// TIA Portal V20 export
DATA_BLOCK "DB_LoaderAxis"   // DB206
// stored: AutoNumber false, InstanceOfName FB_LoaderAxis, InstanceOfType FB
"FB_LoaderAxis"
   // VAR_INPUT
   //    iPLCModeReq : Bool;
   //    iCNCModeReq : Bool;
   //    iU1StartReq : Bool;
   //    iU2StartReq : Bool;
   //    iVStartReq : Bool;
   //    iWStartReq : Bool;
   //    iU1PosSetPoint : Real;
   //    iU2PosSetPoint : Real;
   //    iVPosSetPoint : Real;
   //    iWPosSetPoint : Real;
   // END_VAR
   // VAR_OUTPUT
   //    oU1InPos : Bool;
   //    oU2InPos : Bool;
   //    oVInPos : Bool;
   //    oWInPos : Bool;
   // END_VAR
   // VAR
   //    sAxisPLCMode : Bool;
   //    sAxisCNCMode : Bool;
   //    sAllAxisPLCMode : Bool;
   //    sAllAxisCNCMode : Bool;
   //    sU1StartMove : Bool;
   //    sU2StartMove : Bool;
   //    sVStartMove : Bool;
   //    sWStartMove : Bool;
   //    sU1MoveError : Bool;
   //    sU2MoveError : Bool;
   //    sVMoveError : Bool;
   //    sWMoveError : Bool;
   //    sU1InPos : Bool;
   //    sU2InPos : Bool;
   //    sVInPos : Bool;
   //    sWInPos : Bool;
   //    sU1SetPos : Real;
   //    sU2SetPos : Real;
   //    sVSetPos : Real;
   //    sWSetPos : Real;
   //    sU1MoveState : Byte;
   //    sU2MoveState : Byte;
   //    sVMoveState : Byte;
   //    sWMoveState : Byte;
   //    sU1ActFeedRate : LReal;
   //    sU2ActFeedRate : LReal;
   //    sVActFeedRate : LReal;
   //    sWActFeedRate : LReal;
   //    sU1DrivedByPLC : Bool;
   //    sU2DrivedByPLC : Bool;
   //    sVDrivedByPLC : Bool;
   //    sWDrivedByPLC : Bool;
   //    sU1Positioning { ExternalAccessible := 'False'; ExternalVisible := 'False'; ExternalWritable := 'False'} : Bool;
   //    sU2Positioning { ExternalAccessible := 'False'; ExternalVisible := 'False'; ExternalWritable := 'False'} : Bool;
   //    sVPositioning { ExternalAccessible := 'False'; ExternalVisible := 'False'; ExternalWritable := 'False'} : Bool;
   //    sWPositioning { ExternalAccessible := 'False'; ExternalVisible := 'False'; ExternalWritable := 'False'} : Bool;
   //    sFeedActive : Bool;
   // END_VAR
BEGIN
END_DATA_BLOCK
